{attribute 'qualified_only'}
{attribute 'strict'}
{attribute 'to_string'}
TYPE E_ServiceInternalCommandState :
(
	None := 0,
	Queued := 1,
	RequestHigh := 2,
	Accepted := 3,
	Rejected := 4,
	Cancelled := 5
) UDINT;
END_TYPE

(* stored: Version 1.1.0.1, ProductVersion 3.1.4026.18
   DUT E_ServiceInternalCommandState: Id {38da17c5-93e9-4107-ac63-7a487b3195b8} *)
